ABB RobotStudio station: Ejercicio1_Entregable.rsstnx

Station Ejercicio1_Entregable (saved by RobotStudio 23.2.10395.0)
Controller Controlador
  mechanical unit ROB_1: IRB120_3_58__01, 6 joints, base frame (0, 0, 0) mm
Layout (positions relative to the parent item):
  - Tool_Ej1 [mechanism, from Components\Tool_Ej1.rslib] at (374.67, 11.07, 654.05) mm, rotated rx -176.93 ry 40.2 rz 179.02 deg
  - IRB120_3_58__01 [mechanism, from %ABB.RobotStudio.Models.IRB120%\IRB120_3_58_G_01.rslib] at (0, 0, 0) mm; joint values [0.0478, 0.2269, -0.5261, -0.1036, 1.1739, 0.09] (rad or m)
Attachment: Tool_Ej1 is attached to IRB120_3_58__01 / Link6
Targets, tools, work objects and paths stored in the station, written as RAPID:
! task T_ROB1
MODULE CalibData
  PERS tooldata Tool_Ej1:=[TRUE,[[-90,0,153],[1,0,0,0]],[0.2,[0,0,1],[1,0,0,0],0,0,0]];
ENDMODULE

